Staubli VAL3: Queue.dtx

public num nPush
public num nPop
public num nElems
public MotionCmd buffer[10]
  [0]
    mdesc mDesc = {leave=0, reach=0}
    num nDuration
    num nSequence
    num nMoveType
    jointRx jJointRx
    pointRx pPointRx
  [1]
    mdesc mDesc = {leave=0, reach=0}
    num nDuration
    num nSequence
    num nMoveType
    jointRx jJointRx
    pointRx pPointRx
  [2]
    mdesc mDesc = {leave=0, reach=0}
    num nDuration
    num nSequence
    num nMoveType
    jointRx jJointRx
    pointRx pPointRx
  [3]
    mdesc mDesc = {leave=0, reach=0}
    num nDuration
    num nSequence
    num nMoveType
    jointRx jJointRx
    pointRx pPointRx
  [4]
    mdesc mDesc = {leave=0, reach=0}
    num nDuration
    num nSequence
    num nMoveType
    jointRx jJointRx
    pointRx pPointRx
  [5]
    mdesc mDesc = {leave=0, reach=0}
    num nDuration
    num nSequence
    num nMoveType
    jointRx jJointRx
    pointRx pPointRx
  [6]
    mdesc mDesc = {leave=0, reach=0}
    num nDuration
    num nSequence
    num nMoveType
    jointRx jJointRx
    pointRx pPointRx
  [7]
    mdesc mDesc = {leave=0, reach=0}
    num nDuration
    num nSequence
    num nMoveType
    jointRx jJointRx
    pointRx pPointRx
  [8]
    mdesc mDesc = {leave=0, reach=0}
    num nDuration
    num nSequence
    num nMoveType
    jointRx jJointRx
    pointRx pPointRx
  [9]
    mdesc mDesc = {leave=0, reach=0}
    num nDuration
    num nSequence
    num nMoveType
    jointRx jJointRx
    pointRx pPointRx
